FUNCTION CheckRangeInt : INT
VAR_INPUT
    valueint : INT;
END_VAR

VAR CONSTANT
lowerBound : INT := 0;
upperBound : INT := 32767;
END_VAR

// Controleer of de waarde binnen het bereik ligt en corrigeer deze indien nodig
IF valueint < lowerBound THEN
    CheckRangeInt := lowerBound;
ELSIF valueint > upperBound THEN
    CheckRangeInt := upperBound;
ELSE
    CheckRangeInt := valueint;
END_IF

END_FUNCTION

(* stored: Version 1.1.0.1, ProductVersion 3.1.4024.12
   POU CheckRangeInt: Id {671a4ee4-995e-428d-a46f-3e1a866399a6}, SpecialFunc None *)
